FUNCTION_BLOCK REAL2INT (* Basic Function Block Type *)
  (* Standard: 61499-2 *)
  (* Version 0.0, 7/4/2026, Schneider Electric, Template *)
  PACKAGE SE.Nereda;
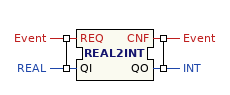
  EVENT_INPUT
    REQ WITH QI; (* Normal Execution Request *)
  END_EVENT
  EVENT_OUTPUT
    CNF WITH QO; (* Execution Confirmation *)
  END_EVENT
  VAR_INPUT
    QI : REAL; (* Input event qualifier *)
  END_VAR
  VAR_OUTPUT
    QO : INT; (* Output event qualifier *)
  END_VAR
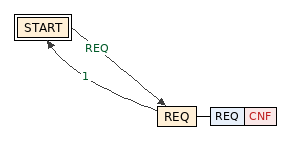
  EC_STATES
    START; (* Initial State *)
    REQ : REQ -> CNF; (* Normal execution *)
  END_STATES
  EC_TRANSITIONS
    START TO REQ := REQ;
    REQ TO START := 1;
  END_TRANSITIONS
  ALGORITHM REQ IN ST: (* Normally executed algorithm *)
(* Conversao REAL -> INT com saturacao: valores fora da faixa do INT
   nao podem chegar ao REAL_TO_INT (erro ERR_RT_CONVERSION para o recurso). *)
IF QI >= 32767.0 THEN
    QO := 32767;
ELSIF QI <= -32768.0 THEN
    QO := -32768;
ELSE
    QO := REAL_TO_INT(QI);
END_IF;
  END_ALGORITHM
END_FUNCTION_BLOCK
